// TwinCAT 3 PLC project OC
// ProgramVersion: 3.1.4026.23
// libraries:
//   OC_Core, * (Open Commissioning)
//   Tc2_Math, * (Beckhoff Automation GmbH)
//   Tc2_Standard, * (Beckhoff Automation GmbH)
//   Tc2_System, * (Beckhoff Automation GmbH)
//   Tc2_Utilities, * (Beckhoff Automation GmbH)
//   Tc3_Module, * (Beckhoff Automation GmbH)
// project tree:
//   FG_01/ FG_01.TcPOU
//   FG_02/ FG_02.TcPOU
//   FG_03/ FG_03.TcPOU
//   FG_04/ FG_04.TcPOU (not stored)
//   FG_05/ FG_05.TcPOU
//   FG_System/ FG_System.TcPOU
//   FG_Transport/ FG_Transport.TcPOU
//   / MAIN.TcPOU, PlcTask.TcTTO (not stored)
//   Sil/PLC/ GVL_PLC.TcGVL, ST_PLCInputs.TcDUT, ST_PLCOutputs.TcDUT
// real-time tasks:
//   TASK PlcTask: cycle T#1ms, priority 4, ADS port 350

// ---- Sil/PLC/ST_PLCInputs.TcDUT
{attribute 'pack_mode' := '0'}
TYPE ST_PLCInputs :
STRUCT
	I0: BYTE;
	I1: BYTE;
	I2: BYTE;
	I3: BYTE;
	I4: BYTE;
	I5: BYTE;
	I6: BYTE;
	I7: BYTE;
	I8: BYTE;
	I9: BYTE;
	I10: BYTE;
	I11: BYTE;
	I12: BYTE;
	I13: BYTE;
	I14: BYTE;
	I15: BYTE;
	I16: BYTE;
	I17: BYTE;
	I18: BYTE;
	I19: BYTE;
	I20: BYTE;
	I21: BYTE;
	I22: BYTE;
	I23: BYTE;
	I24: BYTE;
	I25: BYTE;
	I26: BYTE;
	I27: BYTE;
	I28: BYTE;
	I29: BYTE;
	I30: BYTE;
	I31: BYTE;
	I32: BYTE;
	I33: BYTE;
	I34: BYTE;
	I35: BYTE;
	I36: BYTE;
	I37: BYTE;
	I38: BYTE;
	I39: BYTE;
	I40: BYTE;
	I41: BYTE;
	I42: BYTE;
	I43: BYTE;
	I44: BYTE;
	I45: BYTE;
	I46: BYTE;
	I47: BYTE;
	I48: BYTE;
	I49: BYTE;
	I50: BYTE;
	I51: BYTE;
	I52: BYTE;
	I53: BYTE;
	I54: BYTE;
	I55: BYTE;
	I56: BYTE;
	I57: BYTE;
	I58: BYTE;
	I59: BYTE;
	I60: BYTE;
	I61: BYTE;
	I62: BYTE;
	I63: BYTE;
	I64: BYTE;
	I65: BYTE;
	I66: BYTE;
	I67: BYTE;
	I68: BYTE;
	I69: BYTE;
	I70: BYTE;
	I71: BYTE;
	I72: BYTE;
	I73: BYTE;
	I74: BYTE;
	I75: BYTE;
	I76: BYTE;
	I77: BYTE;
	I78: BYTE;
	I79: BYTE;
	I80: BYTE;
	I81: BYTE;
	I82: BYTE;
	I83: BYTE;
	I84: BYTE;
	I85: BYTE;
	I86: BYTE;
	I87: BYTE;
	I88: BYTE;
	I89: BYTE;
	I90: BYTE;
	I91: BYTE;
	I92: BYTE;
	I93: BYTE;
	I94: BYTE;
	I95: BYTE;
	I96: BYTE;
	I97: BYTE;
	I98: BYTE;
	I99: BYTE;
	I100: BYTE;
	I101: BYTE;
	I102: BYTE;
	I103: BYTE;
	I104: BYTE;
	I105: BYTE;
	I106: BYTE;
	I107: BYTE;
	I108: BYTE;
	I109: BYTE;
	I110: BYTE;
	I111: BYTE;
	I112: BYTE;
	I113: BYTE;
	I114: BYTE;
	I115: BYTE;
	I116: BYTE;
	I117: BYTE;
	I118: BYTE;
	I119: BYTE;
	I120: BYTE;
	I121: BYTE;
	I122: BYTE;
	I123: BYTE;
	I124: BYTE;
	I125: BYTE;
	I126: BYTE;
	I127: BYTE;
	I128: BYTE;
	I129: BYTE;
	I130: BYTE;
	I131: BYTE;
	I132: BYTE;
	I133: BYTE;
	I134: BYTE;
	I135: BYTE;
	I136: BYTE;
	I137: BYTE;
	I138: BYTE;
	I139: BYTE;
	I140: BYTE;
	I141: BYTE;
	I142: BYTE;
	I143: BYTE;
	I144: BYTE;
	I145: BYTE;
	I146: BYTE;
	I147: BYTE;
	I148: BYTE;
	I149: BYTE;
	I150: BYTE;
	I151: BYTE;
	I152: BYTE;
	I153: BYTE;
	I154: BYTE;
	I155: BYTE;
	I156: BYTE;
	I157: BYTE;
	I158: BYTE;
	I159: BYTE;
	I160: BYTE;
	I161: BYTE;
	I162: BYTE;
	I163: BYTE;
	I164: BYTE;
	I165: BYTE;
	I166: BYTE;
	I167: BYTE;
	I168: BYTE;
	I169: BYTE;
	I170: BYTE;
	I171: BYTE;
	I172: BYTE;
	I173: BYTE;
	I174: BYTE;
	I175: BYTE;
	I176: BYTE;
	I177: BYTE;
	I178: BYTE;
	I179: BYTE;
	I180: BYTE;
	I181: BYTE;
	I182: BYTE;
	I183: BYTE;
	I184: BYTE;
	I185: BYTE;
	I186: BYTE;
	I187: BYTE;
	I188: BYTE;
	I189: BYTE;
	I190: BYTE;
	I191: BYTE;
	I192: BYTE;
	I193: BYTE;
	I194: BYTE;
	I195: BYTE;
	I196: BYTE;
	I197: BYTE;
	I198: BYTE;
	I199: BYTE;
	I200: BYTE;
	I201: BYTE;
	I202: BYTE;
	I203: BYTE;
	I204: BYTE;
	I205: BYTE;
	I206: BYTE;
	I207: BYTE;
	I208: BYTE;
	I209: BYTE;
	I210: BYTE;
	I211: BYTE;
	I212: BYTE;
	I213: BYTE;
	I214: BYTE;
	I215: BYTE;
	I216: BYTE;
	I217: BYTE;
	I218: BYTE;
	I219: BYTE;
	I220: BYTE;
	I221: BYTE;
	I222: BYTE;
	I223: BYTE;
	I224: BYTE;
	I225: BYTE;
	I226: BYTE;
	I227: BYTE;
	I228: BYTE;
	I229: BYTE;
	I230: BYTE;
	I231: BYTE;
	I232: BYTE;
	I233: BYTE;
	I234: BYTE;
	I235: BYTE;
	I236: BYTE;
	I237: BYTE;
	I238: BYTE;
	I239: BYTE;
	I240: BYTE;
	I241: BYTE;
	I242: BYTE;
	I243: BYTE;
	I244: BYTE;
	I245: BYTE;
	I246: BYTE;
	I247: BYTE;
	I248: BYTE;
	I249: BYTE;
	I250: BYTE;
	I251: BYTE;
	I252: BYTE;
	I253: BYTE;
	I254: BYTE;
	I255: BYTE;
	I256: BYTE;
	I257: BYTE;
	I258: BYTE;
	I259: BYTE;
	I260: BYTE;
	I261: BYTE;
	I262: BYTE;
	I263: BYTE;
	I264: BYTE;
	I265: BYTE;
	I266: BYTE;
	I267: BYTE;
	I268: BYTE;
	I269: BYTE;
	I270: BYTE;
	I271: BYTE;
	I272: BYTE;
	I273: BYTE;
	I274: BYTE;
	I275: BYTE;
	I276: BYTE;
	I277: BYTE;
	I278: BYTE;
	I279: BYTE;
	I280: BYTE;
	I281: BYTE;
	I282: BYTE;
	I283: BYTE;
	I284: BYTE;
	I285: BYTE;
	I286: BYTE;
	I287: BYTE;
	I288: BYTE;
	I289: BYTE;
	I290: BYTE;
	I291: BYTE;
	I292: BYTE;
	I293: BYTE;
	I294: BYTE;
	I295: BYTE;
	I296: BYTE;
	I297: BYTE;
	I298: BYTE;
	I299: BYTE;
	I300: BYTE;
	I301: BYTE;
	I302: BYTE;
	I303: BYTE;
	I304: BYTE;
	I305: BYTE;
	I306: BYTE;
	I307: BYTE;
	I308: BYTE;
	I309: BYTE;
	I310: BYTE;
	I311: BYTE;
	I312: BYTE;
	I313: BYTE;
	I314: BYTE;
	I315: BYTE;
	I316: BYTE;
	I317: BYTE;
	I318: BYTE;
	I319: BYTE;
	I320: BYTE;
	I321: BYTE;
	I322: BYTE;
	I323: BYTE;
	I324: BYTE;
	I325: BYTE;
	I326: BYTE;
	I327: BYTE;
	I328: BYTE;
	I329: BYTE;
	I330: BYTE;
	I331: BYTE;
	I332: BYTE;
	I333: BYTE;
	I334: BYTE;
	I335: BYTE;
	I336: BYTE;
	I337: BYTE;
	I338: BYTE;
	I339: BYTE;
	I340: BYTE;
	I341: BYTE;
	I342: BYTE;
	I343: BYTE;
	I344: BYTE;
	I345: BYTE;
	I346: BYTE;
	I347: BYTE;
	I348: BYTE;
	I349: BYTE;
	I350: BYTE;
	I351: BYTE;
	I352: BYTE;
	I353: BYTE;
	I354: BYTE;
	I355: BYTE;
	I356: BYTE;
	I357: BYTE;
	I358: BYTE;
	I359: BYTE;
	I360: BYTE;
	I361: BYTE;
	I362: BYTE;
	I363: BYTE;
	I364: BYTE;
	I365: BYTE;
	I366: BYTE;
	I367: BYTE;
	I368: BYTE;
	I369: BYTE;
	I370: BYTE;
	I371: BYTE;
	I372: BYTE;
	I373: BYTE;
	I374: BYTE;
	I375: BYTE;
	I376: BYTE;
	I377: BYTE;
	I378: BYTE;
	I379: BYTE;
	I380: BYTE;
	I381: BYTE;
	I382: BYTE;
	I383: BYTE;
	I384: BYTE;
	I385: BYTE;
	I386: BYTE;
	I387: BYTE;
	I388: BYTE;
	I389: BYTE;
	I390: BYTE;
	I391: BYTE;
	I392: BYTE;
	I393: BYTE;
	I394: BYTE;
	I395: BYTE;
	I396: BYTE;
	I397: BYTE;
	I398: BYTE;
	I399: BYTE;
	I400: BYTE;
	I401: BYTE;
	I402: BYTE;
	I403: BYTE;
	I404: BYTE;
	I405: BYTE;
	I406: BYTE;
	I407: BYTE;
	I408: BYTE;
	I409: BYTE;
	I410: BYTE;
	I411: BYTE;
	I412: BYTE;
	I413: BYTE;
	I414: BYTE;
	I415: BYTE;
	I416: BYTE;
	I417: BYTE;
	I418: BYTE;
	I419: BYTE;
	I420: BYTE;
	I421: BYTE;
	I422: BYTE;
	I423: BYTE;
	I424: BYTE;
	I425: BYTE;
	I426: BYTE;
	I427: BYTE;
	I428: BYTE;
	I429: BYTE;
	I430: BYTE;
	I431: BYTE;
	I432: BYTE;
	I433: BYTE;
	I434: BYTE;
	I435: BYTE;
	I436: BYTE;
	I437: BYTE;
	I438: BYTE;
	I439: BYTE;
	I440: BYTE;
	I441: BYTE;
	I442: BYTE;
	I443: BYTE;
	I444: BYTE;
	I445: BYTE;
	I446: BYTE;
	I447: BYTE;
	I448: BYTE;
	I449: BYTE;
	I450: BYTE;
	I451: BYTE;
	I452: BYTE;
	I453: BYTE;
	I454: BYTE;
	I455: BYTE;
	I456: BYTE;
	I457: BYTE;
	I458: BYTE;
	I459: BYTE;
	I460: BYTE;
	I461: BYTE;
	I462: BYTE;
	I463: BYTE;
	I464: BYTE;
	I465: BYTE;
	I466: BYTE;
	I467: BYTE;
	I468: BYTE;
	I469: BYTE;
	I470: BYTE;
	I471: BYTE;
	I472: BYTE;
	I473: BYTE;
	I474: BYTE;
	I475: BYTE;
	I476: BYTE;
	I477: BYTE;
	I478: BYTE;
	I479: BYTE;
	I480: BYTE;
	I481: BYTE;
	I482: BYTE;
	I483: BYTE;
	I484: BYTE;
	I485: BYTE;
	I486: BYTE;
	I487: BYTE;
	I488: BYTE;
	I489: BYTE;
	I490: BYTE;
	I491: BYTE;
	I492: BYTE;
	I493: BYTE;
	I494: BYTE;
	I495: BYTE;
	I496: BYTE;
	I497: BYTE;
	I498: BYTE;
	I499: BYTE;
	I500: BYTE;
	I501: BYTE;
	I502: BYTE;
	I503: BYTE;
	I504: BYTE;
	I505: BYTE;
	I506: BYTE;
	I507: BYTE;
	I508: BYTE;
	I509: BYTE;
	I510: BYTE;
	I511: BYTE;
	I512: BYTE;
	I513: BYTE;
	I514: BYTE;
	I515: BYTE;
	I516: BYTE;
	I517: BYTE;
	I518: BYTE;
	I519: BYTE;
	I520: BYTE;
	I521: BYTE;
	I522: BYTE;
	I523: BYTE;
	I524: BYTE;
	I525: BYTE;
	I526: BYTE;
	I527: BYTE;
	I528: BYTE;
	I529: BYTE;
	I530: BYTE;
	I531: BYTE;
	I532: BYTE;
	I533: BYTE;
	I534: BYTE;
	I535: BYTE;
	I536: BYTE;
	I537: BYTE;
	I538: BYTE;
	I539: BYTE;
	I540: BYTE;
	I541: BYTE;
	I542: BYTE;
	I543: BYTE;
	I544: BYTE;
	I545: BYTE;
	I546: BYTE;
	I547: BYTE;
	I548: BYTE;
	I549: BYTE;
	I550: BYTE;
	I551: BYTE;
	I552: BYTE;
	I553: BYTE;
	I554: BYTE;
	I555: BYTE;
	I556: BYTE;
	I557: BYTE;
	I558: BYTE;
	I559: BYTE;
	I560: BYTE;
	I561: BYTE;
	I562: BYTE;
	I563: BYTE;
	I564: BYTE;
	I565: BYTE;
	I566: BYTE;
	I567: BYTE;
	I568: BYTE;
	I569: BYTE;
	I570: BYTE;
	I571: BYTE;
	I572: BYTE;
	I573: BYTE;
	I574: BYTE;
	I575: BYTE;
	I576: BYTE;
	I577: BYTE;
	I578: BYTE;
	I579: BYTE;
	I580: BYTE;
	I581: BYTE;
	I582: BYTE;
	I583: BYTE;
	I584: BYTE;
	I585: BYTE;
	I586: BYTE;
	I587: BYTE;
	I588: BYTE;
	I589: BYTE;
	I590: BYTE;
	I591: BYTE;
	I592: BYTE;
	I593: BYTE;
	I594: BYTE;
	I595: BYTE;
	I596: BYTE;
	I597: BYTE;
	I598: BYTE;
	I599: BYTE;
	I600: BYTE;
	I601: BYTE;
	I602: BYTE;
	I603: BYTE;
	I604: BYTE;
	I605: BYTE;
	I606: BYTE;
	I607: BYTE;
	I608: BYTE;
	I609: BYTE;
	I610: BYTE;
	I611: BYTE;
	I612: BYTE;
	I613: BYTE;
	I614: BYTE;
	I615: BYTE;
	I616: BYTE;
	I617: BYTE;
	I618: BYTE;
	I619: BYTE;
	I620: BYTE;
	I621: BYTE;
	I622: BYTE;
	I623: BYTE;
	I624: BYTE;
	I625: BYTE;
	I626: BYTE;
	I627: BYTE;
	I628: BYTE;
	I629: BYTE;
	I630: BYTE;
	I631: BYTE;
	I632: BYTE;
	I633: BYTE;
	I634: BYTE;
	I635: BYTE;
	I636: BYTE;
	I637: BYTE;
	I638: BYTE;
	I639: BYTE;
	I640: BYTE;
	I641: BYTE;
	I642: BYTE;
	I643: BYTE;
	I644: BYTE;
	I645: BYTE;
	I646: BYTE;
	I647: BYTE;
	I648: BYTE;
	I649: BYTE;
	I650: BYTE;
	I651: BYTE;
	I652: BYTE;
	I653: BYTE;
	I654: BYTE;
	I655: BYTE;
	I656: BYTE;
	I657: BYTE;
	I658: BYTE;
	I659: BYTE;
	I660: BYTE;
	I661: BYTE;
	I662: BYTE;
	I663: BYTE;
	I664: BYTE;
	I665: BYTE;
	I666: BYTE;
	I667: BYTE;
	I668: BYTE;
	I669: BYTE;
	I670: BYTE;
	I671: BYTE;
	I672: BYTE;
	I673: BYTE;
	I674: BYTE;
	I675: BYTE;
	I676: BYTE;
	I677: BYTE;
	I678: BYTE;
	I679: BYTE;
	I680: BYTE;
	I681: BYTE;
	I682: BYTE;
	I683: BYTE;
	I684: BYTE;
	I685: BYTE;
	I686: BYTE;
	I687: BYTE;
	I688: BYTE;
	I689: BYTE;
	I690: BYTE;
	I691: BYTE;
	I692: BYTE;
	I693: BYTE;
	I694: BYTE;
	I695: BYTE;
	I696: BYTE;
	I697: BYTE;
	I698: BYTE;
	I699: BYTE;
	I700: BYTE;
	I701: BYTE;
	I702: BYTE;
	I703: BYTE;
	I704: BYTE;
	I705: BYTE;
	I706: BYTE;
	I707: BYTE;
	I708: BYTE;
	I709: BYTE;
	I710: BYTE;
	I711: BYTE;
	I712: BYTE;
	I713: BYTE;
	I714: BYTE;
	I715: BYTE;
	I716: BYTE;
	I717: BYTE;
	I718: BYTE;
	I719: BYTE;
	I720: BYTE;
	I721: BYTE;
	I722: BYTE;
	I723: BYTE;
	I724: BYTE;
	I725: BYTE;
	I726: BYTE;
	I727: BYTE;
	I728: BYTE;
	I729: BYTE;
	I730: BYTE;
	I731: BYTE;
	I732: BYTE;
	I733: BYTE;
	I734: BYTE;
	I735: BYTE;
	I736: BYTE;
	I737: BYTE;
	I738: BYTE;
	I739: BYTE;
	I740: BYTE;
	I741: BYTE;
	I742: BYTE;
	I743: BYTE;
	I744: BYTE;
	I745: BYTE;
	I746: BYTE;
	I747: BYTE;
	I748: BYTE;
	I749: BYTE;
	I750: BYTE;
	I751: BYTE;
	I752: BYTE;
	I753: BYTE;
	I754: BYTE;
	I755: BYTE;
	I756: BYTE;
	I757: BYTE;
	I758: BYTE;
	I759: BYTE;
	I760: BYTE;
	I761: BYTE;
	I762: BYTE;
	I763: BYTE;
	I764: BYTE;
	I765: BYTE;
	I766: BYTE;
	I767: BYTE;
	I768: BYTE;
	I769: BYTE;
	I770: BYTE;
	I771: BYTE;
	I772: BYTE;
	I773: BYTE;
	I774: BYTE;
	I775: BYTE;
	I776: BYTE;
	I777: BYTE;
	I778: BYTE;
	I779: BYTE;
	I780: BYTE;
	I781: BYTE;
	I782: BYTE;
	I783: BYTE;
	I784: BYTE;
	I785: BYTE;
	I786: BYTE;
	I787: BYTE;
	I788: BYTE;
	I789: BYTE;
	I790: BYTE;
	I791: BYTE;
	I792: BYTE;
	I793: BYTE;
	I794: BYTE;
	I795: BYTE;
	I796: BYTE;
	I797: BYTE;
	I798: BYTE;
	I799: BYTE;
	I800: BYTE;
	I801: BYTE;
	I802: BYTE;
	I803: BYTE;
	I804: BYTE;
	I805: BYTE;
	I806: BYTE;
	I807: BYTE;
	I808: BYTE;
	I809: BYTE;
	I810: BYTE;
	I811: BYTE;
	I812: BYTE;
	I813: BYTE;
	I814: BYTE;
	I815: BYTE;
	I816: BYTE;
	I817: BYTE;
	I818: BYTE;
	I819: BYTE;
	I820: BYTE;
	I821: BYTE;
	I822: BYTE;
	I823: BYTE;
	I824: BYTE;
	I825: BYTE;
	I826: BYTE;
	I827: BYTE;
	I828: BYTE;
	I829: BYTE;
	I830: BYTE;
	I831: BYTE;
	I832: BYTE;
	I833: BYTE;
	I834: BYTE;
	I835: BYTE;
	I836: BYTE;
	I837: BYTE;
	I838: BYTE;
	I839: BYTE;
	I840: BYTE;
	I841: BYTE;
	I842: BYTE;
	I843: BYTE;
	I844: BYTE;
	I845: BYTE;
	I846: BYTE;
	I847: BYTE;
	I848: BYTE;
	I849: BYTE;
	I850: BYTE;
	I851: BYTE;
	I852: BYTE;
	I853: BYTE;
	I854: BYTE;
	I855: BYTE;
	I856: BYTE;
	I857: BYTE;
	I858: BYTE;
	I859: BYTE;
	I860: BYTE;
	I861: BYTE;
	I862: BYTE;
	I863: BYTE;
	I864: BYTE;
	I865: BYTE;
	I866: BYTE;
	I867: BYTE;
	I868: BYTE;
	I869: BYTE;
	I870: BYTE;
	I871: BYTE;
	I872: BYTE;
	I873: BYTE;
	I874: BYTE;
	I875: BYTE;
	I876: BYTE;
	I877: BYTE;
	I878: BYTE;
	I879: BYTE;
	I880: BYTE;
	I881: BYTE;
	I882: BYTE;
	I883: BYTE;
	I884: BYTE;
	I885: BYTE;
	I886: BYTE;
	I887: BYTE;
	I888: BYTE;
	I889: BYTE;
	I890: BYTE;
	I891: BYTE;
	I892: BYTE;
	I893: BYTE;
	I894: BYTE;
	I895: BYTE;
	I896: BYTE;
	I897: BYTE;
	I898: BYTE;
	I899: BYTE;
	I900: BYTE;
	I901: BYTE;
	I902: BYTE;
	I903: BYTE;
	I904: BYTE;
	I905: BYTE;
	I906: BYTE;
	I907: BYTE;
	I908: BYTE;
	I909: BYTE;
	I910: BYTE;
	I911: BYTE;
	I912: BYTE;
	I913: BYTE;
	I914: BYTE;
	I915: BYTE;
	I916: BYTE;
	I917: BYTE;
	I918: BYTE;
	I919: BYTE;
	I920: BYTE;
	I921: BYTE;
	I922: BYTE;
	I923: BYTE;
	I924: BYTE;
	I925: BYTE;
	I926: BYTE;
	I927: BYTE;
	I928: BYTE;
	I929: BYTE;
	I930: BYTE;
	I931: BYTE;
	I932: BYTE;
	I933: BYTE;
	I934: BYTE;
	I935: BYTE;
	I936: BYTE;
	I937: BYTE;
	I938: BYTE;
	I939: BYTE;
	I940: BYTE;
	I941: BYTE;
	I942: BYTE;
	I943: BYTE;
	I944: BYTE;
	I945: BYTE;
	I946: BYTE;
	I947: BYTE;
	I948: BYTE;
	I949: BYTE;
	I950: BYTE;
	I951: BYTE;
	I952: BYTE;
	I953: BYTE;
	I954: BYTE;
	I955: BYTE;
	I956: BYTE;
	I957: BYTE;
	I958: BYTE;
	I959: BYTE;
	I960: BYTE;
	I961: BYTE;
	I962: BYTE;
	I963: BYTE;
	I964: BYTE;
	I965: BYTE;
	I966: BYTE;
	I967: BYTE;
	I968: BYTE;
	I969: BYTE;
	I970: BYTE;
	I971: BYTE;
	I972: BYTE;
	I973: BYTE;
	I974: BYTE;
	I975: BYTE;
	I976: BYTE;
	I977: BYTE;
	I978: BYTE;
	I979: BYTE;
	I980: BYTE;
	I981: BYTE;
	I982: BYTE;
	I983: BYTE;
	I984: BYTE;
	I985: BYTE;
	I986: BYTE;
	I987: BYTE;
	I988: BYTE;
	I989: BYTE;
	I990: BYTE;
	I991: BYTE;
	I992: BYTE;
	I993: BYTE;
	I994: BYTE;
	I995: BYTE;
	I996: BYTE;
	I997: BYTE;
	I998: BYTE;
	I999: BYTE;
	I1000: BYTE;
	I1001: BYTE;
	I1002: BYTE;
	I1003: BYTE;
	I1004: BYTE;
	I1005: BYTE;
	I1006: BYTE;
	I1007: BYTE;
	I1008: BYTE;
	I1009: BYTE;
	I1010: BYTE;
	I1011: BYTE;
	I1012: BYTE;
	I1013: BYTE;
	I1014: BYTE;
	I1015: BYTE;
	I1016: BYTE;
	I1017: BYTE;
	I1018: BYTE;
	I1019: BYTE;
	I1020: BYTE;
	I1021: BYTE;
	I1022: BYTE;
	I1023: BYTE;
END_STRUCT
END_TYPE

// ---- Sil/PLC/ST_PLCOutputs.TcDUT
{attribute 'pack_mode' := '0'}
TYPE ST_PLCOutputs :
STRUCT
	Q0: BYTE;
	Q1: BYTE;
	Q2: BYTE;
	Q3: BYTE;
	Q4: BYTE;
	Q5: BYTE;
	Q6: BYTE;
	Q7: BYTE;
	Q8: BYTE;
	Q9: BYTE;
	Q10: BYTE;
	Q11: BYTE;
	Q12: BYTE;
	Q13: BYTE;
	Q14: BYTE;
	Q15: BYTE;
	Q16: BYTE;
	Q17: BYTE;
	Q18: BYTE;
	Q19: BYTE;
	Q20: BYTE;
	Q21: BYTE;
	Q22: BYTE;
	Q23: BYTE;
	Q24: BYTE;
	Q25: BYTE;
	Q26: BYTE;
	Q27: BYTE;
	Q28: BYTE;
	Q29: BYTE;
	Q30: BYTE;
	Q31: BYTE;
	Q32: BYTE;
	Q33: BYTE;
	Q34: BYTE;
	Q35: BYTE;
	Q36: BYTE;
	Q37: BYTE;
	Q38: BYTE;
	Q39: BYTE;
	Q40: BYTE;
	Q41: BYTE;
	Q42: BYTE;
	Q43: BYTE;
	Q44: BYTE;
	Q45: BYTE;
	Q46: BYTE;
	Q47: BYTE;
	Q48: BYTE;
	Q49: BYTE;
	Q50: BYTE;
	Q51: BYTE;
	Q52: BYTE;
	Q53: BYTE;
	Q54: BYTE;
	Q55: BYTE;
	Q56: BYTE;
	Q57: BYTE;
	Q58: BYTE;
	Q59: BYTE;
	Q60: BYTE;
	Q61: BYTE;
	Q62: BYTE;
	Q63: BYTE;
	Q64: BYTE;
	Q65: BYTE;
	Q66: BYTE;
	Q67: BYTE;
	Q68: BYTE;
	Q69: BYTE;
	Q70: BYTE;
	Q71: BYTE;
	Q72: BYTE;
	Q73: BYTE;
	Q74: BYTE;
	Q75: BYTE;
	Q76: BYTE;
	Q77: BYTE;
	Q78: BYTE;
	Q79: BYTE;
	Q80: BYTE;
	Q81: BYTE;
	Q82: BYTE;
	Q83: BYTE;
	Q84: BYTE;
	Q85: BYTE;
	Q86: BYTE;
	Q87: BYTE;
	Q88: BYTE;
	Q89: BYTE;
	Q90: BYTE;
	Q91: BYTE;
	Q92: BYTE;
	Q93: BYTE;
	Q94: BYTE;
	Q95: BYTE;
	Q96: BYTE;
	Q97: BYTE;
	Q98: BYTE;
	Q99: BYTE;
	Q100: BYTE;
	Q101: BYTE;
	Q102: BYTE;
	Q103: BYTE;
	Q104: BYTE;
	Q105: BYTE;
	Q106: BYTE;
	Q107: BYTE;
	Q108: BYTE;
	Q109: BYTE;
	Q110: BYTE;
	Q111: BYTE;
	Q112: BYTE;
	Q113: BYTE;
	Q114: BYTE;
	Q115: BYTE;
	Q116: BYTE;
	Q117: BYTE;
	Q118: BYTE;
	Q119: BYTE;
	Q120: BYTE;
	Q121: BYTE;
	Q122: BYTE;
	Q123: BYTE;
	Q124: BYTE;
	Q125: BYTE;
	Q126: BYTE;
	Q127: BYTE;
	Q128: BYTE;
	Q129: BYTE;
	Q130: BYTE;
	Q131: BYTE;
	Q132: BYTE;
	Q133: BYTE;
	Q134: BYTE;
	Q135: BYTE;
	Q136: BYTE;
	Q137: BYTE;
	Q138: BYTE;
	Q139: BYTE;
	Q140: BYTE;
	Q141: BYTE;
	Q142: BYTE;
	Q143: BYTE;
	Q144: BYTE;
	Q145: BYTE;
	Q146: BYTE;
	Q147: BYTE;
	Q148: BYTE;
	Q149: BYTE;
	Q150: BYTE;
	Q151: BYTE;
	Q152: BYTE;
	Q153: BYTE;
	Q154: BYTE;
	Q155: BYTE;
	Q156: BYTE;
	Q157: BYTE;
	Q158: BYTE;
	Q159: BYTE;
	Q160: BYTE;
	Q161: BYTE;
	Q162: BYTE;
	Q163: BYTE;
	Q164: BYTE;
	Q165: BYTE;
	Q166: BYTE;
	Q167: BYTE;
	Q168: BYTE;
	Q169: BYTE;
	Q170: BYTE;
	Q171: BYTE;
	Q172: BYTE;
	Q173: BYTE;
	Q174: BYTE;
	Q175: BYTE;
	Q176: BYTE;
	Q177: BYTE;
	Q178: BYTE;
	Q179: BYTE;
	Q180: BYTE;
	Q181: BYTE;
	Q182: BYTE;
	Q183: BYTE;
	Q184: BYTE;
	Q185: BYTE;
	Q186: BYTE;
	Q187: BYTE;
	Q188: BYTE;
	Q189: BYTE;
	Q190: BYTE;
	Q191: BYTE;
	Q192: BYTE;
	Q193: BYTE;
	Q194: BYTE;
	Q195: BYTE;
	Q196: BYTE;
	Q197: BYTE;
	Q198: BYTE;
	Q199: BYTE;
	Q200: BYTE;
	Q201: BYTE;
	Q202: BYTE;
	Q203: BYTE;
	Q204: BYTE;
	Q205: BYTE;
	Q206: BYTE;
	Q207: BYTE;
	Q208: BYTE;
	Q209: BYTE;
	Q210: BYTE;
	Q211: BYTE;
	Q212: BYTE;
	Q213: BYTE;
	Q214: BYTE;
	Q215: BYTE;
	Q216: BYTE;
	Q217: BYTE;
	Q218: BYTE;
	Q219: BYTE;
	Q220: BYTE;
	Q221: BYTE;
	Q222: BYTE;
	Q223: BYTE;
	Q224: BYTE;
	Q225: BYTE;
	Q226: BYTE;
	Q227: BYTE;
	Q228: BYTE;
	Q229: BYTE;
	Q230: BYTE;
	Q231: BYTE;
	Q232: BYTE;
	Q233: BYTE;
	Q234: BYTE;
	Q235: BYTE;
	Q236: BYTE;
	Q237: BYTE;
	Q238: BYTE;
	Q239: BYTE;
	Q240: BYTE;
	Q241: BYTE;
	Q242: BYTE;
	Q243: BYTE;
	Q244: BYTE;
	Q245: BYTE;
	Q246: BYTE;
	Q247: BYTE;
	Q248: BYTE;
	Q249: BYTE;
	Q250: BYTE;
	Q251: BYTE;
	Q252: BYTE;
	Q253: BYTE;
	Q254: BYTE;
	Q255: BYTE;
	Q256: BYTE;
	Q257: BYTE;
	Q258: BYTE;
	Q259: BYTE;
	Q260: BYTE;
	Q261: BYTE;
	Q262: BYTE;
	Q263: BYTE;
	Q264: BYTE;
	Q265: BYTE;
	Q266: BYTE;
	Q267: BYTE;
	Q268: BYTE;
	Q269: BYTE;
	Q270: BYTE;
	Q271: BYTE;
	Q272: BYTE;
	Q273: BYTE;
	Q274: BYTE;
	Q275: BYTE;
	Q276: BYTE;
	Q277: BYTE;
	Q278: BYTE;
	Q279: BYTE;
	Q280: BYTE;
	Q281: BYTE;
	Q282: BYTE;
	Q283: BYTE;
	Q284: BYTE;
	Q285: BYTE;
	Q286: BYTE;
	Q287: BYTE;
	Q288: BYTE;
	Q289: BYTE;
	Q290: BYTE;
	Q291: BYTE;
	Q292: BYTE;
	Q293: BYTE;
	Q294: BYTE;
	Q295: BYTE;
	Q296: BYTE;
	Q297: BYTE;
	Q298: BYTE;
	Q299: BYTE;
	Q300: BYTE;
	Q301: BYTE;
	Q302: BYTE;
	Q303: BYTE;
	Q304: BYTE;
	Q305: BYTE;
	Q306: BYTE;
	Q307: BYTE;
	Q308: BYTE;
	Q309: BYTE;
	Q310: BYTE;
	Q311: BYTE;
	Q312: BYTE;
	Q313: BYTE;
	Q314: BYTE;
	Q315: BYTE;
	Q316: BYTE;
	Q317: BYTE;
	Q318: BYTE;
	Q319: BYTE;
	Q320: BYTE;
	Q321: BYTE;
	Q322: BYTE;
	Q323: BYTE;
	Q324: BYTE;
	Q325: BYTE;
	Q326: BYTE;
	Q327: BYTE;
	Q328: BYTE;
	Q329: BYTE;
	Q330: BYTE;
	Q331: BYTE;
	Q332: BYTE;
	Q333: BYTE;
	Q334: BYTE;
	Q335: BYTE;
	Q336: BYTE;
	Q337: BYTE;
	Q338: BYTE;
	Q339: BYTE;
	Q340: BYTE;
	Q341: BYTE;
	Q342: BYTE;
	Q343: BYTE;
	Q344: BYTE;
	Q345: BYTE;
	Q346: BYTE;
	Q347: BYTE;
	Q348: BYTE;
	Q349: BYTE;
	Q350: BYTE;
	Q351: BYTE;
	Q352: BYTE;
	Q353: BYTE;
	Q354: BYTE;
	Q355: BYTE;
	Q356: BYTE;
	Q357: BYTE;
	Q358: BYTE;
	Q359: BYTE;
	Q360: BYTE;
	Q361: BYTE;
	Q362: BYTE;
	Q363: BYTE;
	Q364: BYTE;
	Q365: BYTE;
	Q366: BYTE;
	Q367: BYTE;
	Q368: BYTE;
	Q369: BYTE;
	Q370: BYTE;
	Q371: BYTE;
	Q372: BYTE;
	Q373: BYTE;
	Q374: BYTE;
	Q375: BYTE;
	Q376: BYTE;
	Q377: BYTE;
	Q378: BYTE;
	Q379: BYTE;
	Q380: BYTE;
	Q381: BYTE;
	Q382: BYTE;
	Q383: BYTE;
	Q384: BYTE;
	Q385: BYTE;
	Q386: BYTE;
	Q387: BYTE;
	Q388: BYTE;
	Q389: BYTE;
	Q390: BYTE;
	Q391: BYTE;
	Q392: BYTE;
	Q393: BYTE;
	Q394: BYTE;
	Q395: BYTE;
	Q396: BYTE;
	Q397: BYTE;
	Q398: BYTE;
	Q399: BYTE;
	Q400: BYTE;
	Q401: BYTE;
	Q402: BYTE;
	Q403: BYTE;
	Q404: BYTE;
	Q405: BYTE;
	Q406: BYTE;
	Q407: BYTE;
	Q408: BYTE;
	Q409: BYTE;
	Q410: BYTE;
	Q411: BYTE;
	Q412: BYTE;
	Q413: BYTE;
	Q414: BYTE;
	Q415: BYTE;
	Q416: BYTE;
	Q417: BYTE;
	Q418: BYTE;
	Q419: BYTE;
	Q420: BYTE;
	Q421: BYTE;
	Q422: BYTE;
	Q423: BYTE;
	Q424: BYTE;
	Q425: BYTE;
	Q426: BYTE;
	Q427: BYTE;
	Q428: BYTE;
	Q429: BYTE;
	Q430: BYTE;
	Q431: BYTE;
	Q432: BYTE;
	Q433: BYTE;
	Q434: BYTE;
	Q435: BYTE;
	Q436: BYTE;
	Q437: BYTE;
	Q438: BYTE;
	Q439: BYTE;
	Q440: BYTE;
	Q441: BYTE;
	Q442: BYTE;
	Q443: BYTE;
	Q444: BYTE;
	Q445: BYTE;
	Q446: BYTE;
	Q447: BYTE;
	Q448: BYTE;
	Q449: BYTE;
	Q450: BYTE;
	Q451: BYTE;
	Q452: BYTE;
	Q453: BYTE;
	Q454: BYTE;
	Q455: BYTE;
	Q456: BYTE;
	Q457: BYTE;
	Q458: BYTE;
	Q459: BYTE;
	Q460: BYTE;
	Q461: BYTE;
	Q462: BYTE;
	Q463: BYTE;
	Q464: BYTE;
	Q465: BYTE;
	Q466: BYTE;
	Q467: BYTE;
	Q468: BYTE;
	Q469: BYTE;
	Q470: BYTE;
	Q471: BYTE;
	Q472: BYTE;
	Q473: BYTE;
	Q474: BYTE;
	Q475: BYTE;
	Q476: BYTE;
	Q477: BYTE;
	Q478: BYTE;
	Q479: BYTE;
	Q480: BYTE;
	Q481: BYTE;
	Q482: BYTE;
	Q483: BYTE;
	Q484: BYTE;
	Q485: BYTE;
	Q486: BYTE;
	Q487: BYTE;
	Q488: BYTE;
	Q489: BYTE;
	Q490: BYTE;
	Q491: BYTE;
	Q492: BYTE;
	Q493: BYTE;
	Q494: BYTE;
	Q495: BYTE;
	Q496: BYTE;
	Q497: BYTE;
	Q498: BYTE;
	Q499: BYTE;
	Q500: BYTE;
	Q501: BYTE;
	Q502: BYTE;
	Q503: BYTE;
	Q504: BYTE;
	Q505: BYTE;
	Q506: BYTE;
	Q507: BYTE;
	Q508: BYTE;
	Q509: BYTE;
	Q510: BYTE;
	Q511: BYTE;
	Q512: BYTE;
	Q513: BYTE;
	Q514: BYTE;
	Q515: BYTE;
	Q516: BYTE;
	Q517: BYTE;
	Q518: BYTE;
	Q519: BYTE;
	Q520: BYTE;
	Q521: BYTE;
	Q522: BYTE;
	Q523: BYTE;
	Q524: BYTE;
	Q525: BYTE;
	Q526: BYTE;
	Q527: BYTE;
	Q528: BYTE;
	Q529: BYTE;
	Q530: BYTE;
	Q531: BYTE;
	Q532: BYTE;
	Q533: BYTE;
	Q534: BYTE;
	Q535: BYTE;
	Q536: BYTE;
	Q537: BYTE;
	Q538: BYTE;
	Q539: BYTE;
	Q540: BYTE;
	Q541: BYTE;
	Q542: BYTE;
	Q543: BYTE;
	Q544: BYTE;
	Q545: BYTE;
	Q546: BYTE;
	Q547: BYTE;
	Q548: BYTE;
	Q549: BYTE;
	Q550: BYTE;
	Q551: BYTE;
	Q552: BYTE;
	Q553: BYTE;
	Q554: BYTE;
	Q555: BYTE;
	Q556: BYTE;
	Q557: BYTE;
	Q558: BYTE;
	Q559: BYTE;
	Q560: BYTE;
	Q561: BYTE;
	Q562: BYTE;
	Q563: BYTE;
	Q564: BYTE;
	Q565: BYTE;
	Q566: BYTE;
	Q567: BYTE;
	Q568: BYTE;
	Q569: BYTE;
	Q570: BYTE;
	Q571: BYTE;
	Q572: BYTE;
	Q573: BYTE;
	Q574: BYTE;
	Q575: BYTE;
	Q576: BYTE;
	Q577: BYTE;
	Q578: BYTE;
	Q579: BYTE;
	Q580: BYTE;
	Q581: BYTE;
	Q582: BYTE;
	Q583: BYTE;
	Q584: BYTE;
	Q585: BYTE;
	Q586: BYTE;
	Q587: BYTE;
	Q588: BYTE;
	Q589: BYTE;
	Q590: BYTE;
	Q591: BYTE;
	Q592: BYTE;
	Q593: BYTE;
	Q594: BYTE;
	Q595: BYTE;
	Q596: BYTE;
	Q597: BYTE;
	Q598: BYTE;
	Q599: BYTE;
	Q600: BYTE;
	Q601: BYTE;
	Q602: BYTE;
	Q603: BYTE;
	Q604: BYTE;
	Q605: BYTE;
	Q606: BYTE;
	Q607: BYTE;
	Q608: BYTE;
	Q609: BYTE;
	Q610: BYTE;
	Q611: BYTE;
	Q612: BYTE;
	Q613: BYTE;
	Q614: BYTE;
	Q615: BYTE;
	Q616: BYTE;
	Q617: BYTE;
	Q618: BYTE;
	Q619: BYTE;
	Q620: BYTE;
	Q621: BYTE;
	Q622: BYTE;
	Q623: BYTE;
	Q624: BYTE;
	Q625: BYTE;
	Q626: BYTE;
	Q627: BYTE;
	Q628: BYTE;
	Q629: BYTE;
	Q630: BYTE;
	Q631: BYTE;
	Q632: BYTE;
	Q633: BYTE;
	Q634: BYTE;
	Q635: BYTE;
	Q636: BYTE;
	Q637: BYTE;
	Q638: BYTE;
	Q639: BYTE;
	Q640: BYTE;
	Q641: BYTE;
	Q642: BYTE;
	Q643: BYTE;
	Q644: BYTE;
	Q645: BYTE;
	Q646: BYTE;
	Q647: BYTE;
	Q648: BYTE;
	Q649: BYTE;
	Q650: BYTE;
	Q651: BYTE;
	Q652: BYTE;
	Q653: BYTE;
	Q654: BYTE;
	Q655: BYTE;
	Q656: BYTE;
	Q657: BYTE;
	Q658: BYTE;
	Q659: BYTE;
	Q660: BYTE;
	Q661: BYTE;
	Q662: BYTE;
	Q663: BYTE;
	Q664: BYTE;
	Q665: BYTE;
	Q666: BYTE;
	Q667: BYTE;
	Q668: BYTE;
	Q669: BYTE;
	Q670: BYTE;
	Q671: BYTE;
	Q672: BYTE;
	Q673: BYTE;
	Q674: BYTE;
	Q675: BYTE;
	Q676: BYTE;
	Q677: BYTE;
	Q678: BYTE;
	Q679: BYTE;
	Q680: BYTE;
	Q681: BYTE;
	Q682: BYTE;
	Q683: BYTE;
	Q684: BYTE;
	Q685: BYTE;
	Q686: BYTE;
	Q687: BYTE;
	Q688: BYTE;
	Q689: BYTE;
	Q690: BYTE;
	Q691: BYTE;
	Q692: BYTE;
	Q693: BYTE;
	Q694: BYTE;
	Q695: BYTE;
	Q696: BYTE;
	Q697: BYTE;
	Q698: BYTE;
	Q699: BYTE;
	Q700: BYTE;
	Q701: BYTE;
	Q702: BYTE;
	Q703: BYTE;
	Q704: BYTE;
	Q705: BYTE;
	Q706: BYTE;
	Q707: BYTE;
	Q708: BYTE;
	Q709: BYTE;
	Q710: BYTE;
	Q711: BYTE;
	Q712: BYTE;
	Q713: BYTE;
	Q714: BYTE;
	Q715: BYTE;
	Q716: BYTE;
	Q717: BYTE;
	Q718: BYTE;
	Q719: BYTE;
	Q720: BYTE;
	Q721: BYTE;
	Q722: BYTE;
	Q723: BYTE;
	Q724: BYTE;
	Q725: BYTE;
	Q726: BYTE;
	Q727: BYTE;
	Q728: BYTE;
	Q729: BYTE;
	Q730: BYTE;
	Q731: BYTE;
	Q732: BYTE;
	Q733: BYTE;
	Q734: BYTE;
	Q735: BYTE;
	Q736: BYTE;
	Q737: BYTE;
	Q738: BYTE;
	Q739: BYTE;
	Q740: BYTE;
	Q741: BYTE;
	Q742: BYTE;
	Q743: BYTE;
	Q744: BYTE;
	Q745: BYTE;
	Q746: BYTE;
	Q747: BYTE;
	Q748: BYTE;
	Q749: BYTE;
	Q750: BYTE;
	Q751: BYTE;
	Q752: BYTE;
	Q753: BYTE;
	Q754: BYTE;
	Q755: BYTE;
	Q756: BYTE;
	Q757: BYTE;
	Q758: BYTE;
	Q759: BYTE;
	Q760: BYTE;
	Q761: BYTE;
	Q762: BYTE;
	Q763: BYTE;
	Q764: BYTE;
	Q765: BYTE;
	Q766: BYTE;
	Q767: BYTE;
	Q768: BYTE;
	Q769: BYTE;
	Q770: BYTE;
	Q771: BYTE;
	Q772: BYTE;
	Q773: BYTE;
	Q774: BYTE;
	Q775: BYTE;
	Q776: BYTE;
	Q777: BYTE;
	Q778: BYTE;
	Q779: BYTE;
	Q780: BYTE;
	Q781: BYTE;
	Q782: BYTE;
	Q783: BYTE;
	Q784: BYTE;
	Q785: BYTE;
	Q786: BYTE;
	Q787: BYTE;
	Q788: BYTE;
	Q789: BYTE;
	Q790: BYTE;
	Q791: BYTE;
	Q792: BYTE;
	Q793: BYTE;
	Q794: BYTE;
	Q795: BYTE;
	Q796: BYTE;
	Q797: BYTE;
	Q798: BYTE;
	Q799: BYTE;
	Q800: BYTE;
	Q801: BYTE;
	Q802: BYTE;
	Q803: BYTE;
	Q804: BYTE;
	Q805: BYTE;
	Q806: BYTE;
	Q807: BYTE;
	Q808: BYTE;
	Q809: BYTE;
	Q810: BYTE;
	Q811: BYTE;
	Q812: BYTE;
	Q813: BYTE;
	Q814: BYTE;
	Q815: BYTE;
	Q816: BYTE;
	Q817: BYTE;
	Q818: BYTE;
	Q819: BYTE;
	Q820: BYTE;
	Q821: BYTE;
	Q822: BYTE;
	Q823: BYTE;
	Q824: BYTE;
	Q825: BYTE;
	Q826: BYTE;
	Q827: BYTE;
	Q828: BYTE;
	Q829: BYTE;
	Q830: BYTE;
	Q831: BYTE;
	Q832: BYTE;
	Q833: BYTE;
	Q834: BYTE;
	Q835: BYTE;
	Q836: BYTE;
	Q837: BYTE;
	Q838: BYTE;
	Q839: BYTE;
	Q840: BYTE;
	Q841: BYTE;
	Q842: BYTE;
	Q843: BYTE;
	Q844: BYTE;
	Q845: BYTE;
	Q846: BYTE;
	Q847: BYTE;
	Q848: BYTE;
	Q849: BYTE;
	Q850: BYTE;
	Q851: BYTE;
	Q852: BYTE;
	Q853: BYTE;
	Q854: BYTE;
	Q855: BYTE;
	Q856: BYTE;
	Q857: BYTE;
	Q858: BYTE;
	Q859: BYTE;
	Q860: BYTE;
	Q861: BYTE;
	Q862: BYTE;
	Q863: BYTE;
	Q864: BYTE;
	Q865: BYTE;
	Q866: BYTE;
	Q867: BYTE;
	Q868: BYTE;
	Q869: BYTE;
	Q870: BYTE;
	Q871: BYTE;
	Q872: BYTE;
	Q873: BYTE;
	Q874: BYTE;
	Q875: BYTE;
	Q876: BYTE;
	Q877: BYTE;
	Q878: BYTE;
	Q879: BYTE;
	Q880: BYTE;
	Q881: BYTE;
	Q882: BYTE;
	Q883: BYTE;
	Q884: BYTE;
	Q885: BYTE;
	Q886: BYTE;
	Q887: BYTE;
	Q888: BYTE;
	Q889: BYTE;
	Q890: BYTE;
	Q891: BYTE;
	Q892: BYTE;
	Q893: BYTE;
	Q894: BYTE;
	Q895: BYTE;
	Q896: BYTE;
	Q897: BYTE;
	Q898: BYTE;
	Q899: BYTE;
	Q900: BYTE;
	Q901: BYTE;
	Q902: BYTE;
	Q903: BYTE;
	Q904: BYTE;
	Q905: BYTE;
	Q906: BYTE;
	Q907: BYTE;
	Q908: BYTE;
	Q909: BYTE;
	Q910: BYTE;
	Q911: BYTE;
	Q912: BYTE;
	Q913: BYTE;
	Q914: BYTE;
	Q915: BYTE;
	Q916: BYTE;
	Q917: BYTE;
	Q918: BYTE;
	Q919: BYTE;
	Q920: BYTE;
	Q921: BYTE;
	Q922: BYTE;
	Q923: BYTE;
	Q924: BYTE;
	Q925: BYTE;
	Q926: BYTE;
	Q927: BYTE;
	Q928: BYTE;
	Q929: BYTE;
	Q930: BYTE;
	Q931: BYTE;
	Q932: BYTE;
	Q933: BYTE;
	Q934: BYTE;
	Q935: BYTE;
	Q936: BYTE;
	Q937: BYTE;
	Q938: BYTE;
	Q939: BYTE;
	Q940: BYTE;
	Q941: BYTE;
	Q942: BYTE;
	Q943: BYTE;
	Q944: BYTE;
	Q945: BYTE;
	Q946: BYTE;
	Q947: BYTE;
	Q948: BYTE;
	Q949: BYTE;
	Q950: BYTE;
	Q951: BYTE;
	Q952: BYTE;
	Q953: BYTE;
	Q954: BYTE;
	Q955: BYTE;
	Q956: BYTE;
	Q957: BYTE;
	Q958: BYTE;
	Q959: BYTE;
	Q960: BYTE;
	Q961: BYTE;
	Q962: BYTE;
	Q963: BYTE;
	Q964: BYTE;
	Q965: BYTE;
	Q966: BYTE;
	Q967: BYTE;
	Q968: BYTE;
	Q969: BYTE;
	Q970: BYTE;
	Q971: BYTE;
	Q972: BYTE;
	Q973: BYTE;
	Q974: BYTE;
	Q975: BYTE;
	Q976: BYTE;
	Q977: BYTE;
	Q978: BYTE;
	Q979: BYTE;
	Q980: BYTE;
	Q981: BYTE;
	Q982: BYTE;
	Q983: BYTE;
	Q984: BYTE;
	Q985: BYTE;
	Q986: BYTE;
	Q987: BYTE;
	Q988: BYTE;
	Q989: BYTE;
	Q990: BYTE;
	Q991: BYTE;
	Q992: BYTE;
	Q993: BYTE;
	Q994: BYTE;
	Q995: BYTE;
	Q996: BYTE;
	Q997: BYTE;
	Q998: BYTE;
	Q999: BYTE;
	Q1000: BYTE;
	Q1001: BYTE;
	Q1002: BYTE;
	Q1003: BYTE;
	Q1004: BYTE;
	Q1005: BYTE;
	Q1006: BYTE;
	Q1007: BYTE;
	Q1008: BYTE;
	Q1009: BYTE;
	Q1010: BYTE;
	Q1011: BYTE;
	Q1012: BYTE;
	Q1013: BYTE;
	Q1014: BYTE;
	Q1015: BYTE;
	Q1016: BYTE;
	Q1017: BYTE;
	Q1018: BYTE;
	Q1019: BYTE;
	Q1020: BYTE;
	Q1021: BYTE;
	Q1022: BYTE;
	Q1023: BYTE;
END_STRUCT
END_TYPE

// ---- Sil/PLC/GVL_PLC.TcGVL
{attribute 'linkalways'}
{attribute 'qualified_only'}
{attribute 'subsequent'}
{attribute 'pack_mode' := '1'}
VAR_GLOBAL
	Inputs : ST_PLCInputs;
	Outputs : ST_PLCOutputs;
END_VAR

// ---- FG_01/FG_01.TcPOU
FUNCTION_BLOCK FG_01
{region generated code}
VAR_INPUT
	P_Reader : FB_Reader;
	Y_Gripper : FB_Cylinder;
	Y_LaserMark : FB_DeviceByte;
	Y_Platform : FB_Cylinder;
	Y_ReaderWindow : FB_Cylinder;
END_VAR
{endregion}

{region generated code}
	InitRun();
	P_Reader();
	Y_Gripper();
	Y_LaserMark();
	Y_Platform();
	Y_ReaderWindow();
{endregion}

Mapping();

METHOD InitRun
{region generated code}
VAR_INST
	bInitRun : BOOL := TRUE;
END_VAR
{endregion}
{region generated code}
	IF NOT bInitRun THEN RETURN; END_IF
	bInitRun := FALSE;
{endregion}
END_METHOD

ACTION Mapping:
//Gripper
GVL_PLC.Inputs.I101.0 := Y_Gripper.bRetracted;
GVL_PLC.Inputs.I101.1 := Y_Gripper.bExtended;
Y_Gripper.bExtend 	:= GVL_PLC.Outputs.Q101.1;

//Platform
GVL_PLC.Inputs.I102.0 	:= Y_Platform.bRetracted;
GVL_PLC.Inputs.I102.1 	:= Y_Platform.bExtended;
Y_Platform.bRetract 	:= GVL_PLC.Outputs.Q102.0;
Y_Platform.bExtend 	:= GVL_PLC.Outputs.Q102.1;

//ReaderWindow
GVL_PLC.Inputs.I103.1 	:= Y_ReaderWindow.bExtended;
Y_ReaderWindow.bExtend 	:= GVL_PLC.Outputs.Q103.1;

// TODO: no address in xlsx for P_Reader (FB_Reader)
// TODO: no address in xlsx for Y_LaserMark (FB_DeviceByte)
END_ACTION

END_FUNCTION_BLOCK

// ---- FG_02/FG_02.TcPOU
FUNCTION_BLOCK FG_02
{region generated code}
VAR_INPUT
	H_CameraLight : FB_Lamp;
END_VAR
{endregion}

{region generated code}
	InitRun();
	H_CameraLight();
{endregion}

METHOD InitRun
{region generated code}
VAR_INST
	bInitRun : BOOL := TRUE;
END_VAR
{endregion}
{region generated code}
	IF NOT bInitRun THEN RETURN; END_IF
	bInitRun := FALSE;
{endregion}
END_METHOD

END_FUNCTION_BLOCK

// ---- FG_03/FG_03.TcPOU
FUNCTION_BLOCK FG_03
{region generated code}
VAR_INPUT
	Y_AxisR1 : FB_Cylinder;
	Y_AxisX1 : FB_Cylinder;
	Y_AxisX2 : FB_Cylinder;
	Y_AxisY1 : FB_Cylinder;
	Y_AxisY2 : FB_Cylinder;
	Y_Gripper1 : FB_Cylinder;
	Y_Gripper2 : FB_Cylinder;
END_VAR
{endregion}

{region generated code}
	InitRun();
	Y_AxisR1();
	Y_AxisX1();
	Y_AxisX2();
	Y_AxisY1();
	Y_AxisY2();
	Y_Gripper1();
	Y_Gripper2();
{endregion}

Mapping();

METHOD InitRun
{region generated code}
VAR_INST
	bInitRun : BOOL := TRUE;
END_VAR
{endregion}
{region generated code}
	IF NOT bInitRun THEN RETURN; END_IF
	bInitRun := FALSE;
{endregion}
END_METHOD

ACTION Mapping:
//Axis R1
GVL_PLC.Inputs.I301.0 	:= Y_AxisR1.bRetracted;
GVL_PLC.Inputs.I301.1 	:= Y_AxisR1.bExtended;
Y_AxisR1.bRetract 	:= GVL_PLC.Outputs.Q301.0;
Y_AxisR1.bExtend 	:= GVL_PLC.Outputs.Q301.1;

//Axis X1
GVL_PLC.Inputs.I302.0 	:= Y_AxisX1.bRetracted;
GVL_PLC.Inputs.I302.1 	:= Y_AxisX1.bExtended;
Y_AxisX1.bRetract 	:= GVL_PLC.Outputs.Q302.0;
Y_AxisX1.bExtend 	:= GVL_PLC.Outputs.Q302.1;

//Axis Y1
GVL_PLC.Inputs.I303.0 	:= Y_AxisY1.bRetracted;
GVL_PLC.Inputs.I303.1 	:= Y_AxisY1.bExtended;
Y_AxisY1.bRetract 	:= GVL_PLC.Outputs.Q303.0;
Y_AxisY1.bExtend 	:= GVL_PLC.Outputs.Q303.1;

//Axis X2
GVL_PLC.Inputs.I304.0 	:= Y_AxisX2.bRetracted;
GVL_PLC.Inputs.I304.1 	:= Y_AxisX2.bExtended;
Y_AxisX2.bRetract 	:= GVL_PLC.Outputs.Q304.0;
Y_AxisX2.bExtend 	:= GVL_PLC.Outputs.Q304.1;

//Axis Y2
GVL_PLC.Inputs.I305.0 	:= Y_AxisY2.bRetracted;
GVL_PLC.Inputs.I305.1 	:= Y_AxisY2.bExtended;
Y_AxisY2.bRetract 	:= GVL_PLC.Outputs.Q305.0;
Y_AxisY2.bExtend 	:= GVL_PLC.Outputs.Q305.1;

//Gripper 1
GVL_PLC.Inputs.I306.0 	:= Y_Gripper1.bRetracted;
GVL_PLC.Inputs.I306.1 	:= Y_Gripper1.bExtended;
Y_Gripper1.bRetract 	:= GVL_PLC.Outputs.Q306.0;
Y_Gripper1.bExtend 	:= GVL_PLC.Outputs.Q306.1;

//Gripper 2
GVL_PLC.Inputs.I307.0 	:= Y_Gripper2.bRetracted;
GVL_PLC.Inputs.I307.1 	:= Y_Gripper2.bExtended;
Y_Gripper2.bRetract 	:= GVL_PLC.Outputs.Q307.0;
Y_Gripper2.bExtend 	:= GVL_PLC.Outputs.Q307.1;
END_ACTION

END_FUNCTION_BLOCK

// ---- FG_05/FG_05.TcPOU
FUNCTION_BLOCK FG_05
{region generated code}
VAR_INPUT
	B_Part : FB_SensorBinary;
	P_Camera : FB_Reader;
	Y_AxisR : FB_Cylinder;
	Y_AxisX : FB_Cylinder;
	Y_AxisZ1 : FB_Cylinder;
	Y_AxisZ2 : FB_Cylinder;
	Y_CapsSource : FB_DeviceByte;
	Y_CapsSourceStopper : FB_Cylinder;
	Y_Gripper : FB_Cylinder;
END_VAR
{endregion}

{region generated code}
	InitRun();
	B_Part();
	P_Camera();
	Y_AxisR();
	Y_AxisX();
	Y_AxisZ1();
	Y_AxisZ2();
	Y_CapsSource();
	Y_CapsSourceStopper();
	Y_Gripper();
{endregion}

Mapping();

METHOD InitRun
{region generated code}
VAR_INST
	bInitRun : BOOL := TRUE;
END_VAR
{endregion}
{region generated code}
	IF NOT bInitRun THEN RETURN; END_IF
	bInitRun := FALSE;
{endregion}
END_METHOD

ACTION Mapping:
//Part sensor
GVL_PLC.Inputs.I500.0 	:= B_Part.bValue;

//Axis R
GVL_PLC.Inputs.I501.0 	:= Y_AxisR.bRetracted;
GVL_PLC.Inputs.I501.1 	:= Y_AxisR.bExtended;
Y_AxisR.bRetract 	:= GVL_PLC.Outputs.Q501.0;
Y_AxisR.bExtend 	:= GVL_PLC.Outputs.Q501.1;

//Axis X
GVL_PLC.Inputs.I502.0 	:= Y_AxisX.bRetracted;
GVL_PLC.Inputs.I502.1 	:= Y_AxisX.bExtended;
Y_AxisX.bRetract 	:= GVL_PLC.Outputs.Q502.0;
Y_AxisX.bExtend 	:= GVL_PLC.Outputs.Q502.1;

//Axis Z1
GVL_PLC.Inputs.I503.0 	:= Y_AxisZ1.bRetracted;
GVL_PLC.Inputs.I503.1 	:= Y_AxisZ1.bExtended;
Y_AxisZ1.bRetract 	:= GVL_PLC.Outputs.Q503.0;
Y_AxisZ1.bExtend 	:= GVL_PLC.Outputs.Q503.1;

//Axis Z2
GVL_PLC.Inputs.I504.0 	:= Y_AxisZ2.bRetracted;
GVL_PLC.Inputs.I504.1 	:= Y_AxisZ2.bExtended;
Y_AxisZ2.bRetract 	:= GVL_PLC.Outputs.Q504.0;
Y_AxisZ2.bExtend 	:= GVL_PLC.Outputs.Q504.1;

//Caps Source Stopper
GVL_PLC.Inputs.I505.0 		:= Y_CapsSourceStopper.bRetracted;
Y_CapsSourceStopper.bExtend 	:= GVL_PLC.Outputs.Q505.1;

//Gripper
GVL_PLC.Inputs.I506.0 	:= Y_Gripper.bRetracted;
GVL_PLC.Inputs.I506.1 	:= Y_Gripper.bExtended;
Y_Gripper.bRetract 	:= GVL_PLC.Outputs.Q506.0;
Y_Gripper.bExtend 	:= GVL_PLC.Outputs.Q506.1;

// TODO: no address in xlsx for P_Camera (FB_Reader)
// TODO: no address in xlsx for Y_CapsSource (FB_DeviceByte)
END_ACTION

END_FUNCTION_BLOCK

// ---- FG_System/FG_System.TcPOU
FUNCTION_BLOCK FG_System

{region generated code}
VAR_INPUT
	B_SafetyDoor11 : FB_Lock;
	B_SafetyDoor12 : FB_Lock;
	B_SafetyDoor13 : FB_Lock;
	B_SafetyDoor21 : FB_Lock;
	B_SafetyDoor22 : FB_Lock;
	B_SafetyDoor23 : FB_Lock;
	H_ControlPanel : FB_Panel;
	H_SignalTower : FB_Panel;
	SS_EStop1 : FB_Button;
	SS_EStop2 : FB_Button;
END_VAR
{endregion}

{region generated code}
	InitRun();
	B_SafetyDoor11();
	B_SafetyDoor12();
	B_SafetyDoor13();
	B_SafetyDoor21();
	B_SafetyDoor22();
	B_SafetyDoor23();
	H_ControlPanel();
	H_SignalTower();
	SS_EStop1();
	SS_EStop2();
{endregion}

Mapping();

METHOD InitRun
{region generated code}
VAR_INST
	bInitRun : BOOL := TRUE;
END_VAR
{endregion}
{region generated code}
	IF NOT bInitRun THEN RETURN; END_IF
	bInitRun := FALSE;
{endregion}
END_METHOD

ACTION Mapping:
H_ControlPanel.nControlData.0 := GVL_PLC.Outputs.Q0.1;
H_ControlPanel.nControlData.2 := GVL_PLC.Outputs.Q0.3;
H_ControlPanel.nControlData.3 := GVL_PLC.Outputs.Q0.4;
H_ControlPanel.nControlData.4 := GVL_PLC.Outputs.Q0.5;
H_ControlPanel.nControlData.5 := GVL_PLC.Outputs.Q0.6;
H_ControlPanel.nControlData.6 := GVL_PLC.Outputs.Q0.7;

GVL_PLC.Inputs.I0.1 := H_ControlPanel.nStatusData.0;
GVL_PLC.Inputs.I0.2 := H_ControlPanel.nStatusData.1;
GVL_PLC.Inputs.I0.3 := H_ControlPanel.nStatusData.2;
GVL_PLC.Inputs.I0.4 := H_ControlPanel.nStatusData.3;
GVL_PLC.Inputs.I0.5 := H_ControlPanel.nStatusData.4;
GVL_PLC.Inputs.I0.6 := H_ControlPanel.nStatusData.5;
GVL_PLC.Inputs.I0.7 := H_ControlPanel.nStatusData.6;

H_SignalTower.nControlData.0 := GVL_PLC.Outputs.Q1.2;
H_SignalTower.nControlData.1 := GVL_PLC.Outputs.Q1.1;
H_SignalTower.nControlData.2 := GVL_PLC.Outputs.Q1.0;
END_ACTION

END_FUNCTION_BLOCK

// ---- FG_Transport/FG_Transport.TcPOU
FUNCTION_BLOCK FG_Transport

{region generated code}
VAR_INPUT
	B_SafetyGate1 : FB_SensorBinary;
	B_SafetyGate2 : FB_SensorBinary;
	Index01_B_Detect : FB_SensorBinary;
	Index01_B_Exit : FB_SensorBinary;
	Index01_Y_Lift : FB_Cylinder;
	Index01_Y_Stopper : FB_Cylinder;
	Index02_B_Detect : FB_SensorBinary;
	Index02_B_Exit : FB_SensorBinary;
	Index02_Y_Lift : FB_Cylinder;
	Index02_Y_Stopper : FB_Cylinder;
	Index03_B_Detect : FB_SensorBinary;
	Index03_B_Exit : FB_SensorBinary;
	Index03_Y_Lift : FB_Cylinder;
	Index03_Y_Stopper : FB_Cylinder;
	Index04_B_Detect : FB_SensorBinary;
	Index04_B_Exit : FB_SensorBinary;
	Index04_Y_Lift : FB_Cylinder;
	Index04_Y_Stopper : FB_Cylinder;
	Index05_B_Detect : FB_SensorBinary;
	Index05_B_Exit : FB_SensorBinary;
	Index05_Y_Lift : FB_Cylinder;
	Index05_Y_Stopper : FB_Cylinder;
	Lift01_B_Detect : FB_SensorBinary;
	Lift01_B_Exit : FB_SensorBinary;
	Lift01_M_Conveyor : FB_Drive;
	Lift01_Y_Lift : FB_Cylinder;
	Lift02_B_Detect : FB_SensorBinary;
	Lift02_B_Exit : FB_SensorBinary;
	Lift02_M_Conveyor : FB_Drive;
	Lift02_Y_Lift : FB_Cylinder;
	Stopper01_B_Detect : FB_SensorBinary;
	Stopper01_B_Exit : FB_SensorBinary;
	Stopper01_Y_Stopper : FB_Cylinder;
	Stopper02_B_Detect : FB_SensorBinary;
	Stopper02_B_Exit : FB_SensorBinary;
	Stopper02_Y_Stopper : FB_Cylinder;
	Stopper03_B_Detect : FB_SensorBinary;
	Stopper03_B_Exit : FB_SensorBinary;
	Stopper03_Y_Stopper : FB_Cylinder;
	Stopper04_B_Detect : FB_SensorBinary;
	Stopper04_B_Exit : FB_SensorBinary;
	Stopper04_Y_Stopper : FB_Cylinder;
	Transport01_M_Conveyor : FB_Drive;
	Transport02_M_Conveyor : FB_Drive;
	Y_Gate1 : FB_Cylinder;
	Y_Gate2 : FB_Cylinder;
END_VAR
{endregion}

{region generated code}
	InitRun();
	B_SafetyGate1();
	B_SafetyGate2();
	Index01_B_Detect();
	Index01_B_Exit();
	Index01_Y_Lift();
	Index01_Y_Stopper();
	Index02_B_Detect();
	Index02_B_Exit();
	Index02_Y_Lift();
	Index02_Y_Stopper();
	Index03_B_Detect();
	Index03_B_Exit();
	Index03_Y_Lift();
	Index03_Y_Stopper();
	Index04_B_Detect();
	Index04_B_Exit();
	Index04_Y_Lift();
	Index04_Y_Stopper();
	Index05_B_Detect();
	Index05_B_Exit();
	Index05_Y_Lift();
	Index05_Y_Stopper();
	Lift01_B_Detect();
	Lift01_B_Exit();
	Lift01_M_Conveyor();
	Lift01_Y_Lift();
	Lift02_B_Detect();
	Lift02_B_Exit();
	Lift02_M_Conveyor();
	Lift02_Y_Lift();
	Stopper01_B_Detect();
	Stopper01_B_Exit();
	Stopper01_Y_Stopper();
	Stopper02_B_Detect();
	Stopper02_B_Exit();
	Stopper02_Y_Stopper();
	Stopper03_B_Detect();
	Stopper03_B_Exit();
	Stopper03_Y_Stopper();
	Stopper04_B_Detect();
	Stopper04_B_Exit();
	Stopper04_Y_Stopper();
	Transport01_M_Conveyor();
	Transport02_M_Conveyor();
	Y_Gate1();
	Y_Gate2();
{endregion}

Mapping();

METHOD InitRun
{region generated code}
VAR_INST
	bInitRun : BOOL := TRUE;
END_VAR
{endregion}
{region generated code}
	IF NOT bInitRun THEN RETURN; END_IF
	bInitRun := FALSE;
{endregion}
END_METHOD

ACTION Mapping:
Y_Gate1.bExtend := GVL_PLC.Outputs.Q1001.0;
GVL_PLC.Inputs.I1001.0 := Y_Gate1.bRetracted;
GVL_PLC.Inputs.I1001.1 := Y_Gate1.bExtended;

Y_Gate2.bExtend := GVL_PLC.Outputs.Q1002.0;
GVL_PLC.Inputs.I1002.0 := Y_Gate2.bRetracted;
GVL_PLC.Inputs.I1002.1 := Y_Gate2.bExtended;

//Index Unit 1
GVL_PLC.Inputs.I1003.0 		:= Index01_B_Detect.bValue;
GVL_PLC.Inputs.I1003.1 		:= Index01_B_Exit.bValue;
GVL_PLC.Inputs.I1003.2 		:= Index01_Y_Lift.bRetracted;
GVL_PLC.Inputs.I1003.3 		:= Index01_Y_Lift.bExtended;
GVL_PLC.Inputs.I1003.4 		:= Index01_Y_Stopper.bRetracted;
Index01_Y_Lift.bRetract 	:= GVL_PLC.Outputs.Q1003.0;
Index01_Y_Lift.bExtend 		:= GVL_PLC.Outputs.Q1003.1;
Index01_Y_Stopper.bExtend 	:= GVL_PLC.Outputs.Q1003.2;

//Index Unit 2
GVL_PLC.Inputs.I1004.0 		:= Index02_B_Detect.bValue;
GVL_PLC.Inputs.I1004.1 		:= Index02_B_Exit.bValue;
GVL_PLC.Inputs.I1004.2 		:= Index02_Y_Lift.bRetracted;
GVL_PLC.Inputs.I1004.3 		:= Index02_Y_Lift.bExtended;
GVL_PLC.Inputs.I1004.4 		:= Index02_Y_Stopper.bRetracted;
Index02_Y_Lift.bRetract 	:= GVL_PLC.Outputs.Q1004.0;
Index02_Y_Lift.bExtend 		:= GVL_PLC.Outputs.Q1004.1;
Index02_Y_Stopper.bExtend 	:= GVL_PLC.Outputs.Q1004.2;

//Index Unit 3
GVL_PLC.Inputs.I1005.0 		:= Index03_B_Detect.bValue;
GVL_PLC.Inputs.I1005.1 		:= Index03_B_Exit.bValue;
GVL_PLC.Inputs.I1005.2 		:= Index03_Y_Lift.bRetracted;
GVL_PLC.Inputs.I1005.3 		:= Index03_Y_Lift.bExtended;
GVL_PLC.Inputs.I1005.4 		:= Index03_Y_Stopper.bRetracted;
Index03_Y_Lift.bRetract 	:= GVL_PLC.Outputs.Q1005.0;
Index03_Y_Lift.bExtend 		:= GVL_PLC.Outputs.Q1005.1;
Index03_Y_Stopper.bExtend 	:= GVL_PLC.Outputs.Q1005.2;

//Index Unit 4
GVL_PLC.Inputs.I1006.0 		:= Index04_B_Detect.bValue;
GVL_PLC.Inputs.I1006.1 		:= Index04_B_Exit.bValue;
GVL_PLC.Inputs.I1006.2 		:= Index04_Y_Lift.bRetracted;
GVL_PLC.Inputs.I1006.3 		:= Index04_Y_Lift.bExtended;
GVL_PLC.Inputs.I1006.4 		:= Index04_Y_Stopper.bRetracted;
Index04_Y_Lift.bRetract 	:= GVL_PLC.Outputs.Q1006.0;
Index04_Y_Lift.bExtend 		:= GVL_PLC.Outputs.Q1006.1;
Index04_Y_Stopper.bExtend 	:= GVL_PLC.Outputs.Q1006.2;

//Index Unit 5
GVL_PLC.Inputs.I1007.0 		:= Index05_B_Detect.bValue;
GVL_PLC.Inputs.I1007.1 		:= Index05_B_Exit.bValue;
GVL_PLC.Inputs.I1007.2 		:= Index05_Y_Lift.bRetracted;
GVL_PLC.Inputs.I1007.3 		:= Index05_Y_Lift.bExtended;
GVL_PLC.Inputs.I1007.4 		:= Index05_Y_Stopper.bRetracted;
Index05_Y_Lift.bRetract 	:= GVL_PLC.Outputs.Q1007.0;
Index05_Y_Lift.bExtend 		:= GVL_PLC.Outputs.Q1007.1;
Index05_Y_Stopper.bExtend 	:= GVL_PLC.Outputs.Q1007.2;

//Stopper 1
GVL_PLC.Inputs.I1008.0 		:= Stopper01_B_Detect.bValue;
GVL_PLC.Inputs.I1008.1 		:= Stopper01_B_Exit.bValue;
GVL_PLC.Inputs.I1008.4 		:= Stopper01_Y_Stopper.bRetracted;
Stopper01_Y_Stopper.bExtend	:= GVL_PLC.Outputs.Q1008.2;

//Stopper 2
GVL_PLC.Inputs.I1009.0 		:= Stopper02_B_Detect.bValue;
GVL_PLC.Inputs.I1009.1 		:= Stopper02_B_Exit.bValue;
GVL_PLC.Inputs.I1009.4 		:= Stopper02_Y_Stopper.bRetracted;
Stopper02_Y_Stopper.bExtend	:= GVL_PLC.Outputs.Q1009.2;

//Stopper 3
GVL_PLC.Inputs.I1010.0 		:= Stopper03_B_Detect.bValue;
GVL_PLC.Inputs.I1010.1 		:= Stopper03_B_Exit.bValue;
GVL_PLC.Inputs.I1010.4 		:= Stopper03_Y_Stopper.bRetracted;
Stopper03_Y_Stopper.bExtend	:= GVL_PLC.Outputs.Q1010.2;

//Stopper 4
GVL_PLC.Inputs.I1011.0 		:= Stopper04_B_Detect.bValue;
GVL_PLC.Inputs.I1011.1 		:= Stopper04_B_Exit.bValue;
GVL_PLC.Inputs.I1011.4 		:= Stopper04_Y_Stopper.bRetracted;
Stopper04_Y_Stopper.bExtend	:= GVL_PLC.Outputs.Q1011.2;

//Lift 1
GVL_PLC.Inputs.I1012.0 			:= Lift01_B_Detect.bValue;
GVL_PLC.Inputs.I1012.1 			:= Lift01_B_Exit.bValue;
GVL_PLC.Inputs.I1012.2 			:= Lift01_Y_Lift.bRetracted;
GVL_PLC.Inputs.I1012.3 			:= Lift01_Y_Lift.bExtended;
Lift01_Y_Lift.bRetract 			:= GVL_PLC.Outputs.Q1012.0;
Lift01_Y_Lift.bExtend 			:= GVL_PLC.Outputs.Q1012.1;
Lift01_M_Conveyor.nControl.1 	:= GVL_PLC.Outputs.Q1012.2;
Lift01_M_Conveyor.nControl.0 	:= GVL_PLC.Outputs.Q1012.3;

//Lift 2
GVL_PLC.Inputs.I1013.0 			:= Lift02_B_Detect.bValue;
GVL_PLC.Inputs.I1013.1 			:= Lift02_B_Exit.bValue;
GVL_PLC.Inputs.I1013.2 			:= Lift02_Y_Lift.bRetracted;
GVL_PLC.Inputs.I1013.3 			:= Lift02_Y_Lift.bExtended;
Lift02_Y_Lift.bRetract 			:= GVL_PLC.Outputs.Q1013.0;
Lift02_Y_Lift.bExtend 			:= GVL_PLC.Outputs.Q1013.1;
Lift02_M_Conveyor.nControl.1 	:= GVL_PLC.Outputs.Q1013.2;
Lift02_M_Conveyor.nControl.0 	:= GVL_PLC.Outputs.Q1013.3;

//Transport 1
Transport01_M_Conveyor.nControl.1 	:= GVL_PLC.Outputs.Q1014.0;
Transport01_M_Conveyor.nControl.0 	:= GVL_PLC.Outputs.Q1014.1;

//Transport 2
Transport02_M_Conveyor.nControl.1 	:= GVL_PLC.Outputs.Q1015.0;
Transport02_M_Conveyor.nControl.0 	:= GVL_PLC.Outputs.Q1015.1;
END_ACTION

END_FUNCTION_BLOCK

// ---- MAIN.TcPOU
PROGRAM MAIN

{region generated code}
VAR_INPUT
	bInitRun : BOOL := TRUE;
	fbSystem : FB_System;
	FG_01 : FG_01;
	FG_02 : FG_02;
	FG_03 : FG_03;
	FG_04 : FG_04;
	FG_05 : FG_05;
	FG_System : FG_System;
	FG_Transport : FG_Transport;
END_VAR
{endregion}

{region generated code}
	InitRun();
	fbSystem();
	FG_01();
	FG_02();
	FG_03();
	FG_04();
	FG_05();
	FG_System();
	FG_Transport();
{endregion}

METHOD InitRun
{region generated code}
	IF NOT bInitRun THEN RETURN; END_IF
	bInitRun := FALSE;
{endregion}
END_METHOD

END_PROGRAM
